FUNCTION_BLOCK PID_Regler
VAR_INPUT
	r1 :			REAL;
	y1 :			REAL;
	Modus :		System_Modus_Enum;
	Param :		PID_Parameter_Strukt;
	T :			REAL;
END_VAR
VAR_OUTPUT
	u :			REAL;
END_VAR
VAR
	a0 :		REAL;
	b0 :		REAL;
	c0 :		REAL;

	rm :		REAL;
	ym :		REAL;
	u_temp :	REAL;
	up : 		REAL;
	ui :		REAL;
	ud :		REAL;
	uim :		REAL;
	udm :		REAL;
END_VAR

CASE Modus OF
	System_Modus_Enum.System_Init:
	c0 := (T*Param.Kp)/(2*Param.Ti);
	a0 := (Param.Td)/(Param.Td+Param.N*T);
	b0 := (Param.Kp*Param.Td*Param.N)/(Param.Td+Param.N*T);
	u := 0;
	rm := 0;
	ym := 0;
	up := 0;
	ui := 0;
	ud := 0;
	uim := 0;
	udm := 0;
	;
	System_Modus_Enum.System_Run:
	up := (r1-y1) * Param.Kp;
	IF Param.ARW = TRUE THEN
		ui := uim + c0*((r1-y1)+(rm-ym)) + (T/Param.Tr)*(u-u_temp);
	ELSE
		ui := uim + c0*((r1-y1)+(rm-ym));
	END_IF
	ud := b0 * ((r1-y1)-(rm-ym)) + a0 * udm;
	u := up + ui + ud;
	u_temp := u;
	IF u >= Param.umax THEN
		u := Param.umax;
	END_IF
	IF u <= Param.umin THEN
		u := Param.umin;
	END_IF
	rm := r1;
	ym := y1;
	uim := ui;
	udm := ud;
	;
END_CASE

END_FUNCTION_BLOCK

(* stored: Version 1.1.0.1, ProductVersion 3.1.4024.13
   POU PID_Regler: Id {446a73e7-e224-40d9-96e5-2366c5e9aed5}, SpecialFunc None *)
